% RSLogix 500 project JMP_LBL_Class.RSS, saved by version 8.30.00.16 %
PROJECT "UNTITLED"    % processor: MicroLogix 1000 %

PROGRAM FILES
  LAD 2 "MAIN_PROG"  5 rungs
  LAD 3 "USER_FAULT"  1 rungs
  LAD 4 "HSC_INT"  1 rungs
  LAD 5 "STI_INT"  1 rungs
  LAD 6, 7, 8, 9, 10, 11, 12, 13, 14, 15, 16: only END

DATA FILES
  O0 OUTPUT  1 elements
  I1 INPUT  2 elements
  S2 STATUS  33 elements
  B3 BINARY  32 elements
  T4 TIMER  40 elements
  C5 COUNTER  32 elements
  R6 CONTROL  16 elements
  N7 INTEGER  105 elements

LADDER 2 "MAIN_PROG"
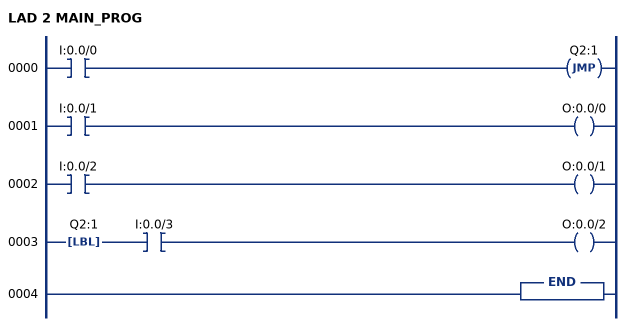
% Rung: 0 %
SOR XIC I:0.0/0 JMP Q2:1 EOR
% Rung: 1 %  % edit flag set %
SOR XIC I:0.0/1 OTE O:0.0/0 EOR
% Rung: 2 %
SOR XIC I:0.0/2 OTE O:0.0/1 EOR
% Rung: 3 %
SOR LBL Q2:1 XIC I:0.0/3 OTE O:0.0/2 EOR
% Rung: 4 %
SOR END EOR
